Fanuc KAREL source: KC00034.KL

PROGRAM KC00034
%NOLOCKGROUP
VAR
  I: INTEGER
  J: INTEGER
  K: INTEGER
  R: REAL
  B: BOOLEAN
  S: STRING[80]
  T: STRING[80]
  P: PATH
  Q: PATH
  AI: ARRAY[8] OF INTEGER
  AB: ARRAY[244] OF BYTE
  F: FILE
BEGIN
  XML_REMTAG(F,S,I)
END KC00034
